FUNCTION_BLOCK New (* _ *)
  (* Version 2015-09-16 *)
END_FUNCTION_BLOCK
(* other elements stored in the file *)
(* SNS LeftPageBorder=-300.0 RightPageBorder=300.0 *)
(* place Diameter=30.0 Name=1 Num=0 LocNum=0 Mark=0 Clock=0 Capacity=1 Comment=_ *)
(* CommentBox Width=20 Height=20 *)
(* place Diameter=30.0 Name=2 Num=1 LocNum=1 Mark=0 Clock=0 Capacity=1 Comment=_ *)
(* CommentBox Width=20 Height=20 *)
(* trans Width=30 Height=20 Num=0 LocNum=0 Name=1 Type=OR TransInscription=_ SwitchMode=s Comment=_ *)
(* CommentBox Width=20 Height=20 *)
(* trans Width=30 Height=20 Num=1 LocNum=1 Name=2 Type=OR TransInscription=_ SwitchMode=s Comment=_ *)
(* CommentBox Width=20 Height=20 *)
(* arc StartPoint=2 EndPoint=1 ArcWeight=1 Comment=_ *)
